// TIA Portal project "Interference" (V15.1)

(* hardware
DEVICE "S7-1200 station_1"  S7-1200 Station
   slot 0: "Rack_0"  S7-1200 Rack  Rack  V1.0
   slot 1: "PLC_1"  CPU 1212C AC/DC/Rly  6ES7 212-1BE40-0XB0  V4.2
*)

// ===== PLC "PLC_1"  CPU 1212C AC/DC/Rly =====

VAR_GLOBAL   // PLC tag table "Default tag table"
   "System_Byte" AT %MB1 : Byte;
   "FirstScan" AT %M1.0 : Bool;
   "DiagStatusUpdate" AT %M1.1 : Bool;
   "AlwaysTRUE" AT %M1.2 : Bool;
   "AlwaysFALSE" AT %M1.3 : Bool;
   "System_Byte(1)" AT %MB1 : Byte;
   "System_Byte(2)" AT %MB1 : Byte;
   "Clock_Byte" AT %MB0 : Byte;
   "Clock_10Hz" AT %M0.0 : Bool;
   "Clock_5Hz" AT %M0.1 : Bool;
   "Clock_2.5Hz" AT %M0.2 : Bool;
   "Clock_2Hz" AT %M0.3 : Bool;
   "Clock_1.25Hz" AT %M0.4 : Bool;
   "Clock_1Hz" AT %M0.5 : Bool;
   "Clock_0.625Hz" AT %M0.6 : Bool;
   "Clock_0.5Hz" AT %M0.7 : Bool;
   "PUT_done" AT %M2.0 : Bool;
   "PUT_Status" AT %MW4 : Word;
   "PUT_error" AT %M2.1 : Bool;
   "Get_done" AT %M2.2 : Bool;
   "GET_Status" AT %MW6 : Word;
   "GET_error" AT %M2.3 : Bool;
END_VAR

DATA_BLOCK "General"   // DB1
{ S7_Optimized_Access := 'TRUE' }
VERSION : 0.1
   VAR
      Send : Bool;
      Recv : Bool;
   END_VAR
BEGIN
END_DATA_BLOCK

DATA_BLOCK "RecvDB"   // DB100
{ S7_Optimized_Access := 'FALSE' }
VERSION : 0.1
BEGIN
END_DATA_BLOCK

DATA_BLOCK "SendDataDB"   // DB200
{ S7_Optimized_Access := 'FALSE' }
VERSION : 0.1
   VAR
      "Bool" : Bool;
      Bool_1 : Bool;
      Bool_2 : Bool;
      Bool_3 : Bool;
      Bool_4 : Bool;
      Bool_5 : Bool;
      Bool_6 : Bool;
      Bool_7 : Bool;
      "INT" : Int;
   END_VAR
BEGIN
END_DATA_BLOCK

ORGANIZATION_BLOCK "Main"   // OB1, LAD, ProgramCycle
TITLE = "Main Program Sweep (Cycle)"
{ S7_Optimized_Access := 'TRUE' }
VERSION : 0.1
   VAR_INPUT
      Initial_Call : Bool;   // Initial call of this OB
      Remanence : Bool;   // =True, if remanent data are available
   END_VAR
   VAR_TEMP   // added for the SCL form of the ladder/FBD networks
      _w1 : Bool;
   END_VAR
BEGIN

REGION Network 1: PUT function
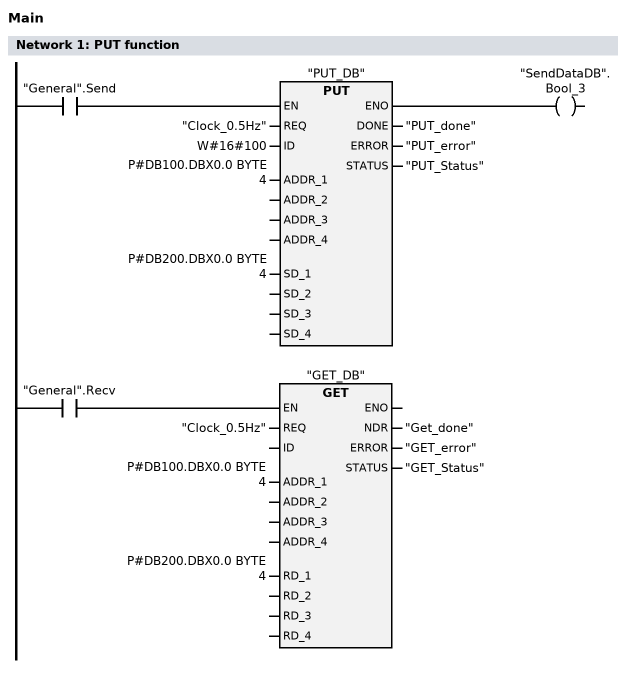
   // ENO of a box is taken as its EN; it also drops when the box reports an error
   #_w1 := "General".Send;
   IF #_w1 THEN
       "PUT_DB"(REQ := "Clock_0.5Hz",   // PUT
                ID := W#16#100,
                ADDR_1 := P#DB100.DBX0.0 BYTE 4,
                SD_1 := P#DB200.DBX0.0 BYTE 4,
                DONE => "PUT_done",
                ERROR => "PUT_error",
                STATUS => "PUT_Status");
   END_IF;
   "SendDataDB".Bool_3 := #_w1;
   IF "General".Recv THEN
       "GET_DB"(REQ := "Clock_0.5Hz",   // GET
                ADDR_1 := P#DB100.DBX0.0 BYTE 4,
                RD_1 := P#DB200.DBX0.0 BYTE 4,
                NDR => "Get_done",
                ERROR => "GET_error",
                STATUS => "GET_Status");
   END_IF;
END_REGION
END_ORGANIZATION_BLOCK